(* PLC project Adressering.ecp, WAGO e!COCKPIT e!COCKPIT *)
(* stored: creationDateTime 2021-01-18T14:20:23.2110188, modificationDateTime 2021-01-18T11:51:27.6823754 *)

TYPE typVAV : STRUCT
  xReady : BOOL;  (* Status adr. *)
  xEnable : BOOL;  (* Enable MP blokk *)
  xAddress : BOOL;  (* Adresserer VAV *)
  xFailed : BOOL;  (* Tilbakemelding adressering (True = SerieNr inn og ut ikke stemmer) *)
  sSetStatus : STRING;  (* Status tilbakemelding naar adresseringen er i SET step *)
  sGetStatus : STRING;  (* Status tilbakemelding naar adresseringen er i GET step *)
  iSerialNr : typSerialNo;  (* Serie NR *)
  bPort : BYTE;  (* VAV Port *)
  bAddress : BYTE;  (* VAV Address *)
  xInitialize : BOOL;  (* initializer tilhoerende vav *)
  rAirVolume_SP : REAL;  (* Settpunkt 0-100% *)
  rOutPosition : REAL;  (* Vinkel *)
  rOutAirVolume_perc : REAL;  (* Luftmengde i prosent *)
  rOutAirVolume_m3h : REAL;  (* Luftmengde i m3h *)
  wSensorValue : WORD;
  rVmin : REAL;
  rVmax : REAL;  (* Max vinkel *)
  xControlRangeIncreased : BOOL;
  xMecanicalOverload : BOOL;
  xActuatorHunting : BOOL;
  xSensorError : BOOL;
  xManualOpen : BOOL;
  xManualClose : BOOL;
  vMin : REAL;  (* Min luftmengde SP / 0-100 *)
  vNorm : REAL;  (* Settpunkt ved bevegelse / 0-100 *)
  vMax : REAL;  (* Maks luftmengde SP / 0-100 *)
  vSize : REAL;  (* Max kubikk *)
  vSetpoint_m3h : REAL;  (* SP% *)
  xdontoptimize : BOOL;  (* Fjerner VAV fra Optimizer *)
END_STRUCT;
END_TYPE

{attribute 'qualified_only'}
VAR_GLOBAL RETAIN PERSISTENT  (* 1.txt *)
  stlv80_a_360_3I302_SQ401 : typVAV := (xEnable := TRUE, vMin := 30, vNorm := 100, vMax := 200, vSize := 434, bPort := 1, bAddress := 1, iSerialNr := (wYearAndWeek := 01945, wDayAndNumber := 20056, bTypeID := 158, bTestStation := 158));  (* / *)
END_VAR

FUNCTION_BLOCK fbAutAd
  VAR_INPUT
    iSerialNr : typSerialNo;
    bPort : BYTE;
    bAddress : BYTE;
    xReset : BOOL;
    xNext : BOOL;
  END_VAR
  VAR_OUTPUT
    i : INT := 0;
    xFailed : BOOL;
    sSetStatus : STRING;
    sGetStatus : STRING;
  END_VAR
  VAR
    xLearn : BOOL;
    xRetry : BOOL;
    VAV_Addressing : fbMpBusAddressing;
    Sleep : TON;
  END_VAR

					//Resetter
IF xReset THEN
	i:= 0;
	xRetry:= FALSE;

//Begynner paa neste VAV
ELSIF i<1 AND xNext THEN
	i:= 1;

//Skriver rett port og adresse til VAV naar blokken er klar
ELSIF VAV_Addressing.xReady AND i=1 AND Sleep.Q THEN
	VAV_Addressing
	(
		xSet:= TRUE,
		xLearn:= xLearn
	);
	i:= 2;
	//Spoer etter serie nr som hoerer til port og adresse
ELSIF VAV_Addressing.xReady AND i=2 AND Sleep.Q THEN
	sSetStatus:= VAV_Addressing.sStatus;
	VAV_Addressing
	(
		xGetSerialNO:= TRUE,
		xLearn:= xLearn
	);
	i:= 3;
	//Sjekker om serie nr. som tilhoerer port og adressen stemmer
ELSIF VAV_Addressing.xReady AND i=3 AND Sleep.Q THEN
	sGetStatus:= VAV_Addressing.sStatus;
	//Sjekker om serie nr stemmer
	IF xRetry AND VAV_Addressing.typOUTSerialNo.wYearAndWeek <> iSerialNr.wYearAndWeek OR VAV_Addressing.typOUTSerialNo.wDayAndNumber <> iSerialNr.wDayAndNumber OR VAV_Addressing.typOUTSerialNo.bTypeID <> iSerialNr.bTypeID OR VAV_Addressing.typOUTSerialNo.bTestStation <> iSerialNr.bTestStation THEN
		xRetry:= FALSE;
		xFailed:= TRUE;
		i:=4;
	ELSIF VAV_Addressing.typOUTSerialNo.wYearAndWeek <> iSerialNr.wYearAndWeek OR VAV_Addressing.typOUTSerialNo.wDayAndNumber <> iSerialNr.wDayAndNumber OR VAV_Addressing.typOUTSerialNo.bTypeID <> iSerialNr.bTypeID OR VAV_Addressing.typOUTSerialNo.bTestStation <> iSerialNr.bTestStation THEN
		xRetry:= TRUE;
		i:=1;
	ELSE
		i:=4;
	END_IF
	Sleep(IN:= FALSE, PT:= T#2S);

//Resetter xSet og xGet, og Setter Port, adresse og serie nr. og henter status

ELSE
	VAV_Addressing
	(
		bPortMpBus:= bPort,
		bAddress:= bAddress,
		typINSerialNo:= iSerialNr,
		xLearn:= xLearn,
		xSet:= FALSE,
		xGetSerialNO:= FALSE,
		xLearn:= xLearn
	);
END_IF
				
END_FUNCTION_BLOCK

PROGRAM PRG_VAV_Adressering
  VAR
    xReset : BOOL;
    xRun : BOOL;
    xInit : BOOL := TRUE;
    Auto : fbAutAd;
    iLinje : INT;  (* Linje som skal adresseres *)
    iVAV : INT := 1;  (* VAV(adr.) som adresseres *)
  END_VAR

					IF xReset THEN
	Auto(xReset:= TRUE);
	xInit:= TRUE;
	xReset:= FALSE;
ELSIF xRun THEN

	IF 1.txt.stlv80_a_360_3I302_SQ401.xAddress OR (iLinje = 1 AND iVAV = 1) THEN

	IF xInit THEN
		1.txt.stlv80_a_360_3I302_SQ401.xEnable:= FALSE;
		Auto(
			bPort:= 1.txt.stlv80_a_360_3I302_SQ401.bPort,
			bAddress:= 1.txt.stlv80_a_360_3I302_SQ401.bAddress,
			iSerialNr:= 1.txt.stlv80_a_360_3I302_SQ401.iSerialNr,
			xNext:= TRUE,
			xReset:= FALSE
			);
		xInit:= FALSE;

	ELSIF Auto.i=4 THEN
		1.txt.stlv80_a_360_3I302_SQ401.sSetStatus:= Auto.sSetStatus;
			1.txt.stlv80_a_360_3I302_SQ401.sGetStatus:= Auto.sGetStatus;
			1.txt.stlv80_a_360_3I302_SQ401.xFailed:= Auto.xFailed;
			1.txt.stlv80_a_360_3I302_SQ401.xAddress:= FALSE;
			1.txt.stlv80_a_360_3I302_SQ401.xEnable:= TRUE;
			xReset:= TRUE;
			iVAV:=iVAV+1;

		ELSE
			Auto(xNext:= FALSE);
		END_IF

	END_IF
END_IF

				
END_PROGRAM
